(* Schneider Machine Expert - Basic project cb, file version 2.6.0.0 *)
(* ProjectInformations: Name=New project *)

HARDWARE
  Cpu 0: TM221CE40R
  EthernetConfiguration: NetworkName=M221, IpAllocationMode=FixedAddress, IpAddress=192.168.0.2, SubnetMask=255.255.255.0
  SerialLineConfiguration: Baud=Baud19200, Parity=ParityEven, DataBits=DataBits8, StopBits=StopBits1, PhysicalMedium=PhysicalMediumRs485, TransmissionMode=TransmissionModeModbusRtu, SlaveId=1, Addressing=SlaveAddressing
  MastTask: UsePeriodScanMode=false, PeriodScan=100
  FastTask: Period=255
  CpuBehavior: StartingMode=StartAsPreviousState, AutoSaveRamOnEeprom=true, WatchdogPeriod=250

SYMBOLS  (address, symbol, comment, settings)
  %M0         "START"
  %M1         "MOVE_TRF"
  %M2         "GRIPPER_C_CLOSE"
  %M3         "MOVE_BACK_TRF"
  %M4         "GRIPPER_ROTATE_CLOSE"
  %M5         "STATUS CB ON"
  %M6         "RELEASE_C_GRIPPER"
  %M7         "POLARITY_ RESULT"
  %M8         "POLARITY_CHECK"
  %M9         "ROTATE_0"
  %M10        "REVERSE_ROTATION"
  %M11        "RESET"
  %M12        "MANUAL"
  %M13        "CB_LF"
  %M14        "CB_RT"
  %M15        "ACTIVE_BOWLFEEDER"
  %M22        "M_Q0"
  %M23        "M_Q1"
  %M24        "M_Q2"
  %M25        "M_Q3"
  %M26        "M_Q4"
  %M27        "M_Q5"
  %M28        "M_Q6"
  %M100       "START GUI"
  %M102       "M_START"
  %I0.0       "EMG"
  %I0.1       "BTN START"
  %I0.2       "LF_CB_FWD"
  %I0.3       "LF_CB_BWD"
  %I0.4       "RT_CB_FWD"
  %I0.5       "RT_CB_BWD"
  %I0.6       "R_0"
  %I0.7       "R_1"
  %I0.8       "GRIP_R_OPEN"
  %I0.9       "GRIP_R_CLOSE"
  %I0.10      "GRIP_C_OPEN"
  %I0.11      "GRIP_C_CLOSE"
  %I0.12      "C_TRF_FWD"
  %I0.13      "TRF_C_BWD"
  %I0.14      "PART_DETECTION"
  %I0.15      "POLARITY"
  %Q0.0       "LF_CB"
  %Q0.1       "RT_CB"
  %Q0.2       "R_P"
  %Q0.3       "GRIP_UPPER"
  %Q0.4       "GRIP_C"
  %Q0.5       "TRF_C"
  %Q0.6       "BOWL_FEEDER"
  %Q0.7       "GRIP_UPPER"

POU New POU
  (* SectionNumber=1 *)

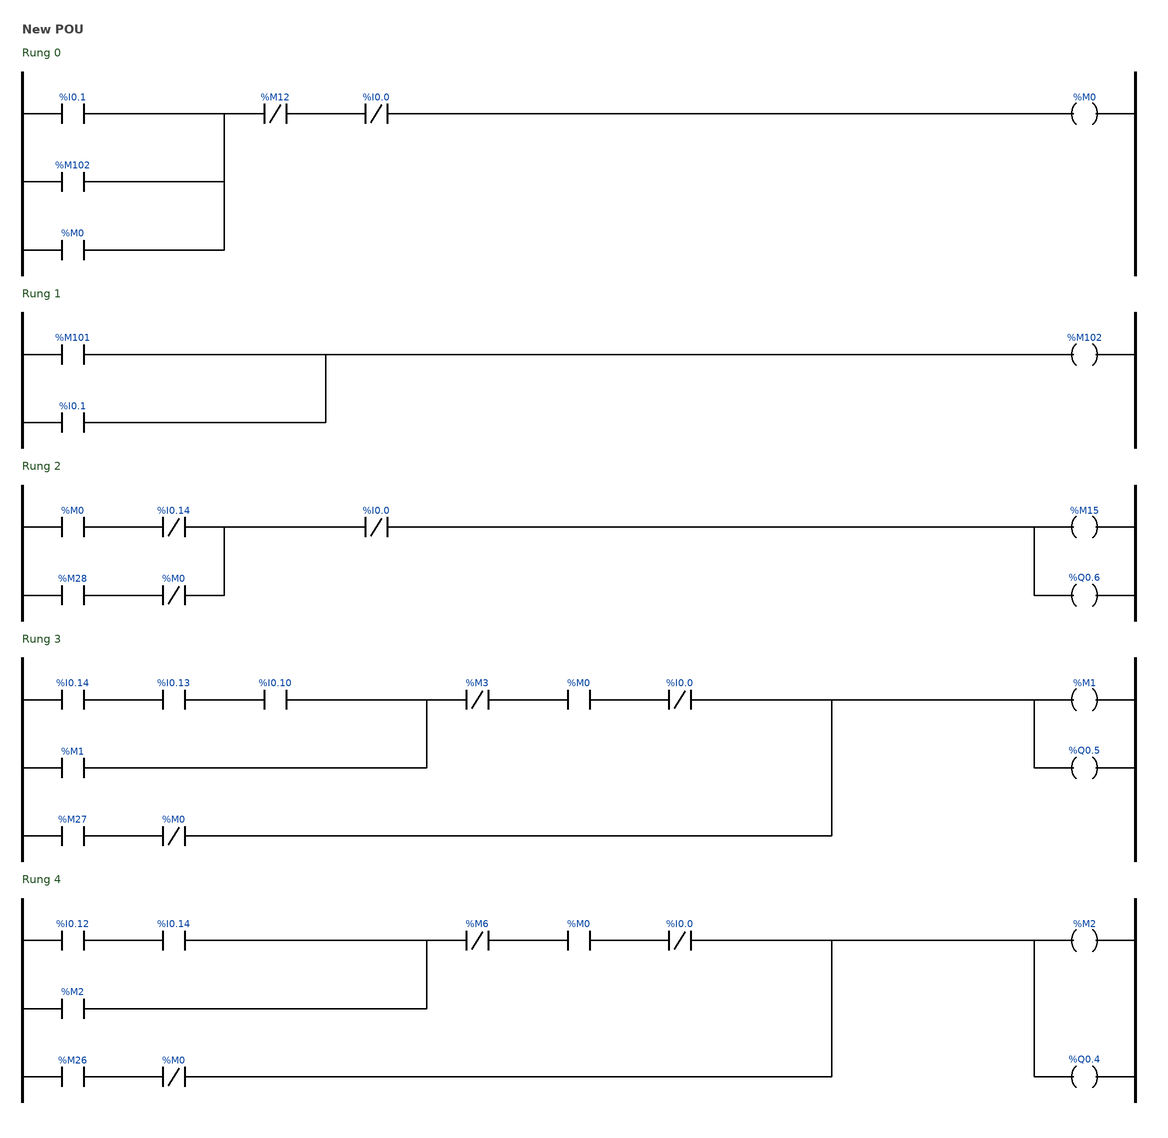

// Rung 0
  LD %I0.1
  OR %M102
  OR %M0
  ANDN %M12
  ANDN %I0.0
  ST %M0
  // as ST:
  //   %M0 := (%I0.1 OR %M102 OR %M0) AND NOT %M12 AND NOT %I0.0;

// Rung 1
  LD %M101
  OR %I0.1
  ST %M102
  // as ST:
  //   %M102 := %M101 OR %I0.1;

// Rung 2
  LD %M0
  ANDN %I0.14
  OR( %M28
  ANDN %M0
  )
  ANDN %I0.0
  ST %M15
  ST %Q0.6
  // as ST:
  //   %M15 := (%M0 AND NOT %I0.14 OR %M28 AND NOT %M0) AND NOT %I0.0;
  //   %Q0.6 := (%M0 AND NOT %I0.14 OR %M28 AND NOT %M0) AND NOT %I0.0;

// Rung 3
  LD %I0.14
  AND %I0.13
  AND %I0.10
  OR %M1
  ANDN %M3
  AND %M0
  ANDN %I0.0
  OR( %M27
  ANDN %M0
  )
  ST %M1
  ST %Q0.5
  // as ST:
  //   _t1 := (%I0.14 AND %I0.13 AND %I0.10 OR %M1) AND NOT %M3 AND %M0 AND NOT %I0.0 OR %M27 AND NOT %M0;
  //   %M1 := _t1;
  //   %Q0.5 := _t1;

// Rung 4
  LD %I0.12
  AND %I0.14
  OR %M2
  ANDN %M6
  AND %M0
  ANDN %I0.0
  OR( %M26
  ANDN %M0
  )
  ST %M2
  ST %Q0.4
  // as ST:
  //   _t1 := (%I0.12 AND %I0.14 OR %M2) AND NOT %M6 AND %M0 AND NOT %I0.0 OR %M26 AND NOT %M0;
  //   %M2 := _t1;
  //   %Q0.4 := _t1;

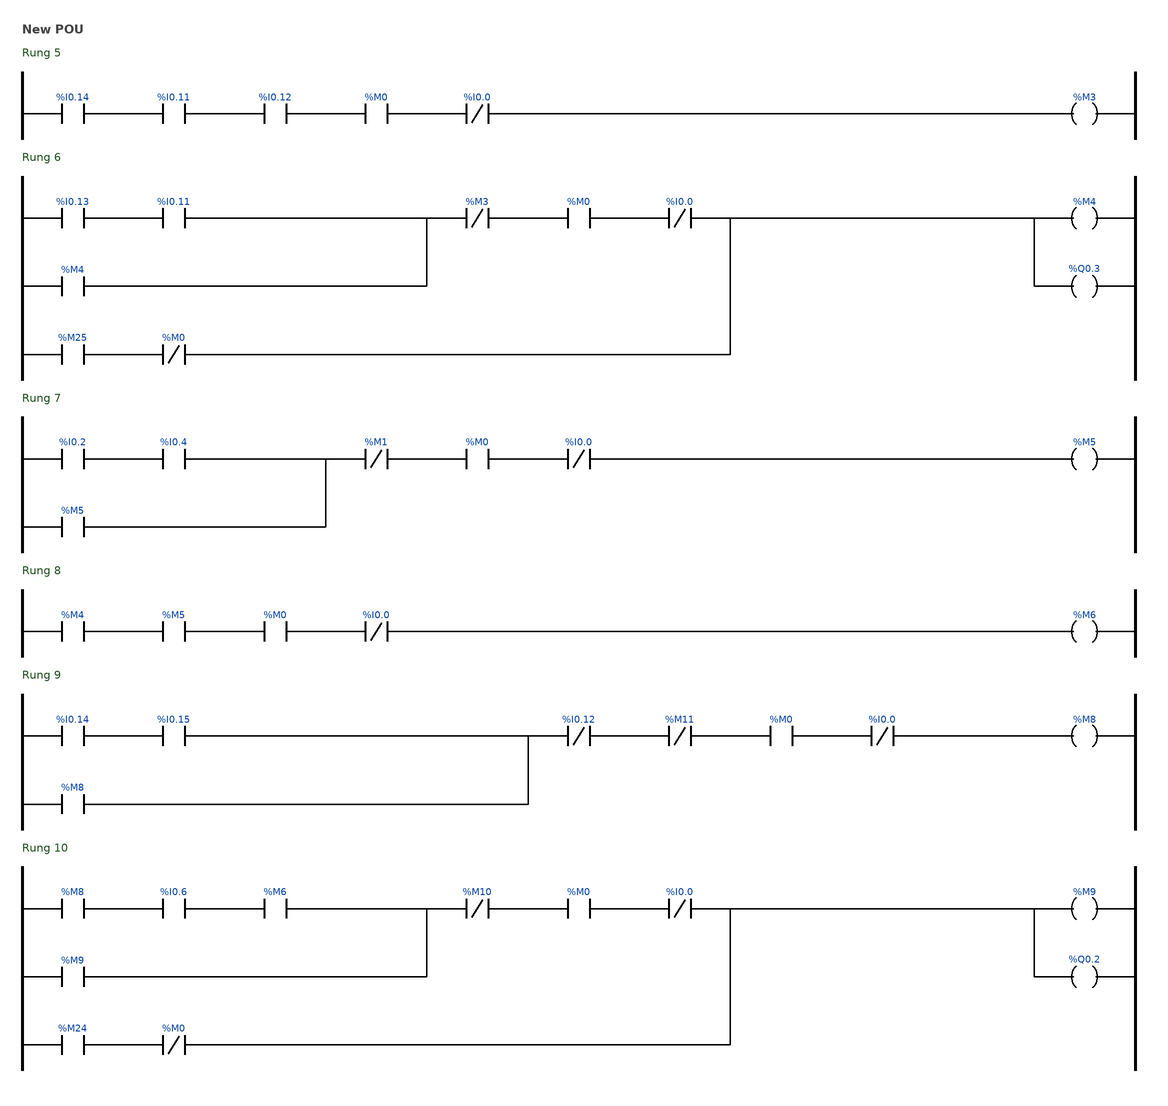

// Rung 5
  LD %I0.14
  AND %I0.11
  AND %I0.12
  AND %M0
  ANDN %I0.0
  ST %M3
  // as ST:
  //   %M3 := %I0.14 AND %I0.11 AND %I0.12 AND %M0 AND NOT %I0.0;

// Rung 6
  LD %I0.13
  AND %I0.11
  OR %M4
  ANDN %M3
  AND %M0
  ANDN %I0.0
  OR( %M25
  ANDN %M0
  )
  ST %M4
  ST %Q0.3
  // as ST:
  //   _t1 := (%I0.13 AND %I0.11 OR %M4) AND NOT %M3 AND %M0 AND NOT %I0.0 OR %M25 AND NOT %M0;
  //   %M4 := _t1;
  //   %Q0.3 := _t1;

// Rung 7
  LD %I0.2
  AND %I0.4
  OR %M5
  ANDN %M1
  AND %M0
  ANDN %I0.0
  ST %M5
  // as ST:
  //   %M5 := (%I0.2 AND %I0.4 OR %M5) AND NOT %M1 AND %M0 AND NOT %I0.0;

// Rung 8
  LD %M4
  AND %M5
  AND %M0
  ANDN %I0.0
  ST %M6
  // as ST:
  //   %M6 := %M4 AND %M5 AND %M0 AND NOT %I0.0;

// Rung 9
  LD %I0.14
  AND %I0.15
  OR %M8
  ANDN %I0.12
  ANDN %M11
  AND %M0
  ANDN %I0.0
  ST %M8
  // as ST:
  //   %M8 := (%I0.14 AND %I0.15 OR %M8) AND NOT %I0.12 AND NOT %M11 AND %M0 AND NOT %I0.0;

// Rung 10
  LD %M8
  AND %I0.6
  AND %M6
  OR %M9
  ANDN %M10
  AND %M0
  ANDN %I0.0
  OR( %M24
  ANDN %M0
  )
  ST %M9
  ST %Q0.2
  // as ST:
  //   _t1 := (%M8 AND %I0.6 AND %M6 OR %M9) AND NOT %M10 AND %M0 AND NOT %I0.0 OR %M24 AND NOT %M0;
  //   %M9 := _t1;
  //   %Q0.2 := _t1;

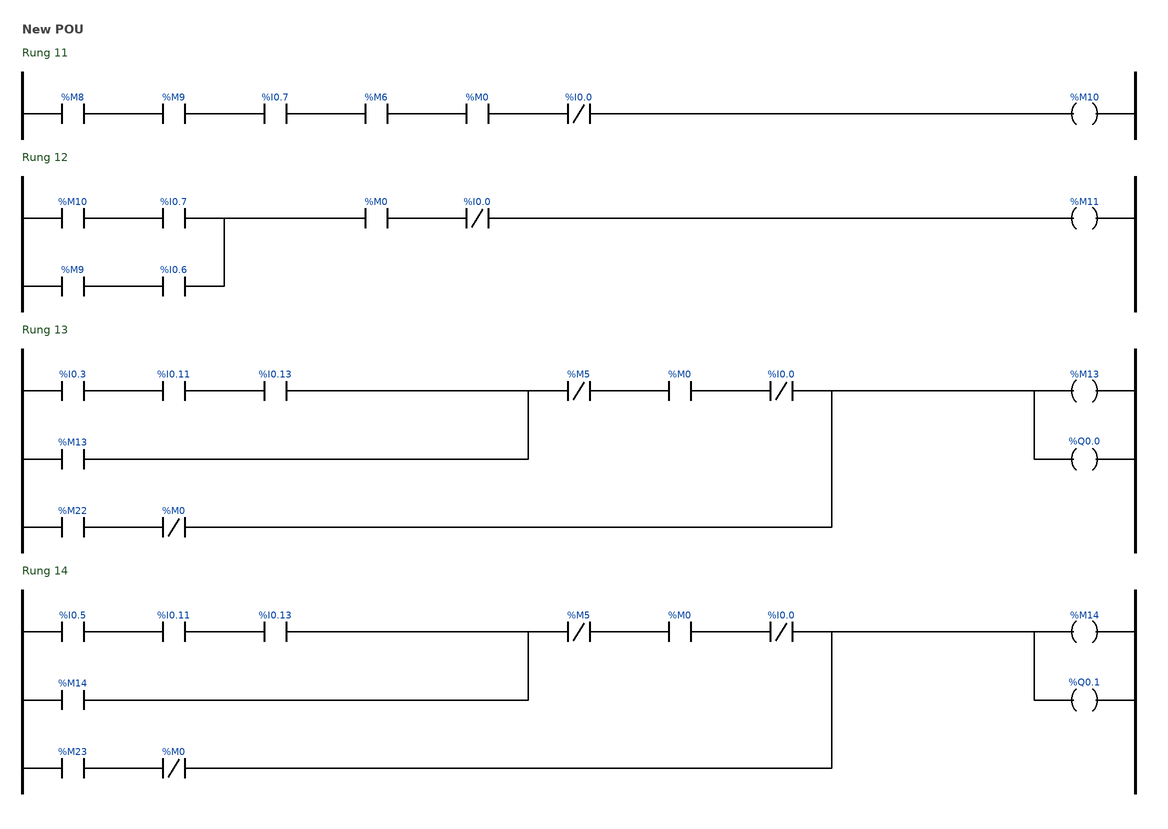

// Rung 11
  LD %M8
  AND %M9
  AND %I0.7
  AND %M6
  AND %M0
  ANDN %I0.0
  ST %M10
  // as ST:
  //   %M10 := %M8 AND %M9 AND %I0.7 AND %M6 AND %M0 AND NOT %I0.0;

// Rung 12
  LD %M10
  AND %I0.7
  OR( %M9
  AND %I0.6
  )
  AND %M0
  ANDN %I0.0
  ST %M11
  // as ST:
  //   %M11 := (%M10 AND %I0.7 OR %M9 AND %I0.6) AND %M0 AND NOT %I0.0;

// Rung 13
  LD %I0.3
  AND %I0.11
  AND %I0.13
  OR %M13
  ANDN %M5
  AND %M0
  ANDN %I0.0
  OR( %M22
  ANDN %M0
  )
  ST %M13
  ST %Q0.0
  // as ST:
  //   _t1 := (%I0.3 AND %I0.11 AND %I0.13 OR %M13) AND NOT %M5 AND %M0 AND NOT %I0.0 OR %M22 AND NOT %M0;
  //   %M13 := _t1;
  //   %Q0.0 := _t1;

// Rung 14
  LD %I0.5
  AND %I0.11
  AND %I0.13
  OR %M14
  ANDN %M5
  AND %M0
  ANDN %I0.0
  OR( %M23
  ANDN %M0
  )
  ST %M14
  ST %Q0.1
  // as ST:
  //   _t1 := (%I0.5 AND %I0.11 AND %I0.13 OR %M14) AND NOT %M5 AND %M0 AND NOT %I0.0 OR %M23 AND NOT %M0;
  //   %M14 := _t1;
  //   %Q0.1 := _t1;

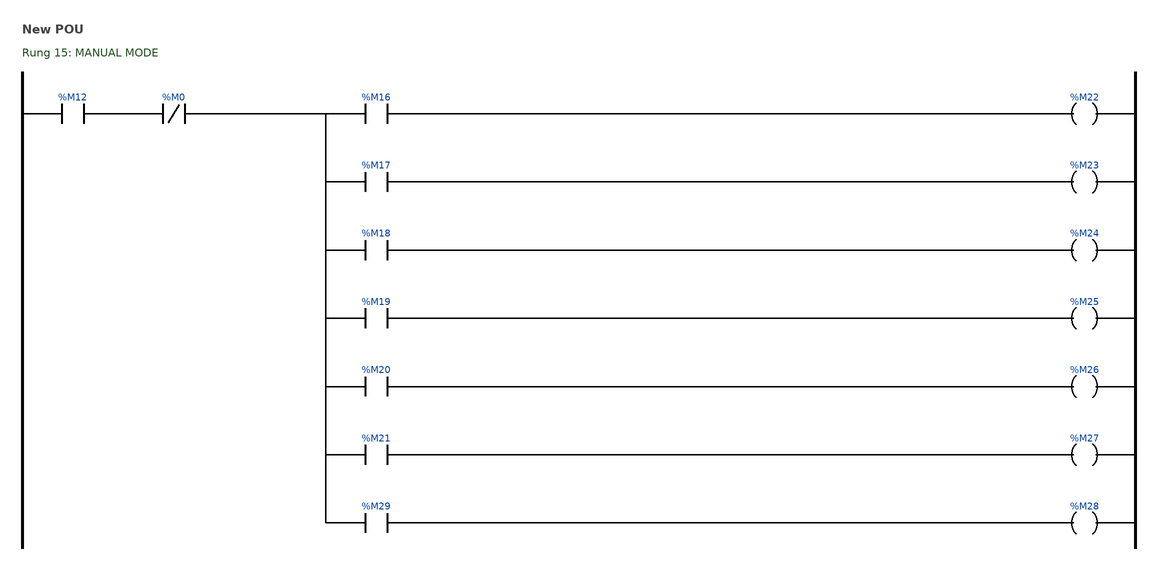

// Rung 15: MANUAL MODE
  LD %M12
  ANDN %M0
  MPS
  AND %M16
  ST %M22
  MRD
  AND %M17
  ST %M23
  MRD
  AND %M18
  ST %M24
  MRD
  AND %M19
  ST %M25
  MRD
  AND %M20
  ST %M26
  MRD
  AND %M21
  ST %M27
  MPP
  AND %M29
  ST %M28
  // as ST:
  //   %M22 := %M12 AND NOT %M0 AND %M16;
  //   %M23 := %M12 AND NOT %M0 AND %M17;
  //   %M24 := %M12 AND NOT %M0 AND %M18;
  //   %M25 := %M12 AND NOT %M0 AND %M19;
  //   %M26 := %M12 AND NOT %M0 AND %M20;
  //   %M27 := %M12 AND NOT %M0 AND %M21;
  //   %M28 := %M12 AND NOT %M0 AND %M29;

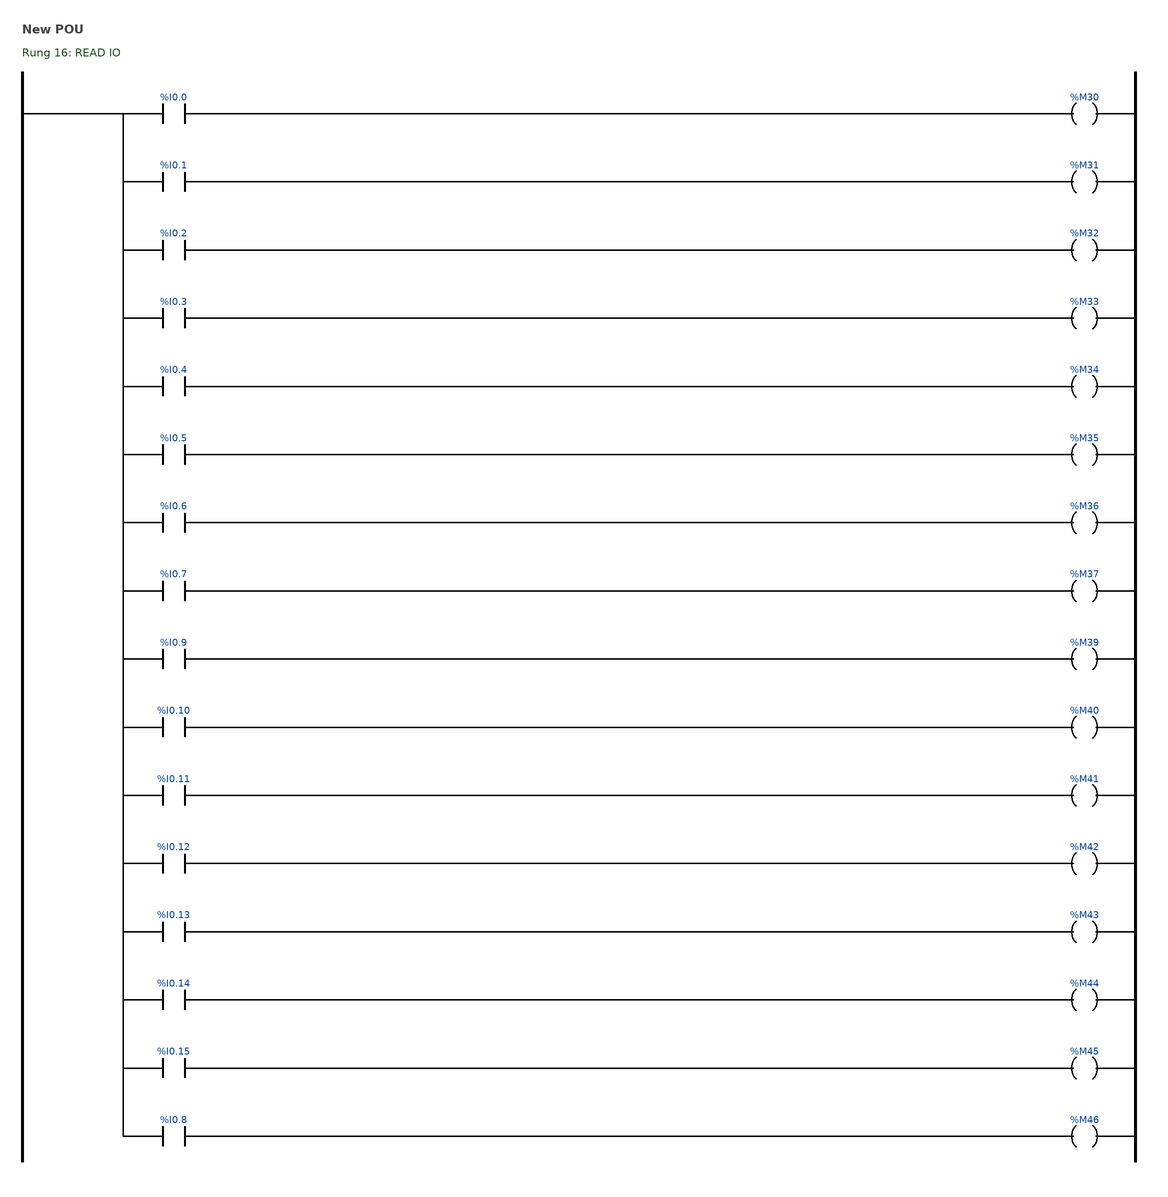

// Rung 16: READ IO
  LD 1
  MPS
  AND %I0.0
  ST %M30
  MRD
  AND %I0.1
  ST %M31
  MRD
  AND %I0.2
  ST %M32
  MRD
  AND %I0.3
  ST %M33
  MRD
  AND %I0.4
  ST %M34
  MRD
  AND %I0.5
  ST %M35
  MRD
  AND %I0.6
  ST %M36
  MRD
  AND %I0.7
  ST %M37
  MRD
  AND %I0.9
  ST %M39
  MRD
  AND %I0.10
  ST %M40
  MRD
  AND %I0.11
  ST %M41
  MRD
  AND %I0.12
  ST %M42
  MRD
  AND %I0.13
  ST %M43
  MRD
  AND %I0.14
  ST %M44
  MRD
  AND %I0.15
  ST %M45
  MPP
  AND %I0.8
  ST %M46
  // as ST:
  //   %M30 := %I0.0;
  //   %M31 := %I0.1;
  //   %M32 := %I0.2;
  //   %M33 := %I0.3;
  //   %M34 := %I0.4;
  //   %M35 := %I0.5;
  //   %M36 := %I0.6;
  //   %M37 := %I0.7;
  //   %M39 := %I0.9;
  //   %M40 := %I0.10;
  //   %M41 := %I0.11;
  //   %M42 := %I0.12;
  //   %M43 := %I0.13;
  //   %M44 := %I0.14;
  //   %M45 := %I0.15;
  //   %M46 := %I0.8;
